Staubli VAL3: connectHostRos.pjx

--- connectHostRos.pjx ---
Parameters version=s7.9.1 stackSize=5000 millimeterUnit=true
Program file=decodeRecvData.pgx
Program file=encodeSendData.pgx
Program file=initTcpIpSocket.pgx
Program file=recvData.pgx
Program file=recvRosMsg.pgx
Program file=sendData.pgx
Program file=sendFbkMsg.pgx
Program file=start.pgx
Program file=stop.pgx
Data file=connectHostRos.dtx
Type name=FlagStatus path=Disk://RobotController_Libs/FlagStatus/FlagStatus.pjx
Type name=RobotStatus path=Disk://RobotController_Libs/RobotStatus/RobotStatus.pjx
Type name=CommParameter path=Disk://RobotController_Libs/CommParameter/CommParameter.pjx

--- connectHostRos.dtx ---
mdesc mNomSpeed
public sio soTcpIpFbk
public sio siTcpIpMotion
public num nRecvData[53]
public CommParameter cRosMotionParm
  [0]
    num port
    string target
    num clients
    num endOfString
    num timeOut
    num baudRate
    string parity
    num bits
    num stopBits
    string mode
    string flowControl
    bool nagle
public CommParameter cRosFbkParm
  [0]
    num port
    string target
    num clients
    num endOfString
    num timeOut
    num baudRate
    string parity
    num bits
    num stopBits
    string mode
    string flowControl
    bool nagle
public FlagStatus fRosStatus
  [0]
    num ForceFlag
    num RosFlag
    num RobotFlag
public num nSendData[52]

--- decodeRecvData.pgx ---
public program decodeRecvData(num& x_nRecvData[], RobotStatus& x_rRobotStatus, FlagStatus& x_fDataStatus, num& x_nRosFlagCmd)
  local num l_nNum
begin

  //This program is used for decoding the received data from host ROS contorlller.

  //suppose the received data containing 1 identifier, 24 joint status 27 cartesian status and 1 ROS flag
  //and ensure the received data intact
  if size(x_nRecvData)==53
    //assert the received ROS massages OK
    x_fDataStatus.RosFlag=1
    //decode the received data to the format of robot controller(Staubli SRS format)
    x_rRobotStatus.jointSpace.JointPos.j1=x_nRecvData[1]
    x_rRobotStatus.jointSpace.JointPos.j2=x_nRecvData[2]
    x_rRobotStatus.jointSpace.JointPos.j3=x_nRecvData[3]
    x_rRobotStatus.jointSpace.JointPos.j4=x_nRecvData[4]
    x_rRobotStatus.jointSpace.JointPos.j5=x_nRecvData[5]
    x_rRobotStatus.jointSpace.JointPos.j6=x_nRecvData[6]

    x_rRobotStatus.cartesianSpace.CartesianPos.trsf.x=x_nRecvData[25]
    x_rRobotStatus.cartesianSpace.CartesianPos.trsf.y=x_nRecvData[26]
    x_rRobotStatus.cartesianSpace.CartesianPos.trsf.z=x_nRecvData[27]
    x_rRobotStatus.cartesianSpace.CartesianPos.trsf.rx=x_nRecvData[28]
    x_rRobotStatus.cartesianSpace.CartesianPos.trsf.ry=x_nRecvData[29]
    x_rRobotStatus.cartesianSpace.CartesianPos.trsf.rz=x_nRecvData[30]

    for l_nNum=0 to 5
      x_rRobotStatus.jointSpace.JointVel[l_nNum]=x_nRecvData[l_nNum+7]
      x_rRobotStatus.jointSpace.JointAccel[l_nNum]=x_nRecvData[l_nNum+13]
      x_rRobotStatus.jointSpace.JointForce[l_nNum]=x_nRecvData[l_nNum+19]

      x_rRobotStatus.cartesianSpace.CartesianVel[l_nNum]=x_nRecvData[l_nNum+31]
      x_rRobotStatus.cartesianSpace.CartesianAccel[l_nNum]=x_nRecvData[l_nNum+37]
      x_rRobotStatus.cartesianSpace.CartesianForce[l_nNum]=x_nRecvData[l_nNum+43]
    endFor

    x_rRobotStatus.cartesianSpace.CarteResVel=x_nRecvData[49]
    x_rRobotStatus.cartesianSpace.CarteResAccel=x_nRecvData[50]
    x_rRobotStatus.cartesianSpace.CarteResForce=x_nRecvData[51]
    x_nRosFlagCmd=x_nRecvData[52]

  else
    x_fDataStatus.RosFlag=-1

  endIf

end

--- encodeSendData.pgx ---
public program encodeSendData(num& x_nSendData[], RobotStatus& x_rRobotStatus)
  local num l_nNum
begin

  //This program is used for encoding the data sent to the host ROS controller.

  //suppose the sent data containing 1 identifier，24 joint status and 27 cartesian status
  //and ensure the sent data intact
  x_nSendData[0]=0

  x_nSendData[1]=x_rRobotStatus.jointSpace.JointPos.j1
  x_nSendData[2]=x_rRobotStatus.jointSpace.JointPos.j2
  x_nSendData[3]=x_rRobotStatus.jointSpace.JointPos.j3
  x_nSendData[4]=x_rRobotStatus.jointSpace.JointPos.j4
  x_nSendData[5]=x_rRobotStatus.jointSpace.JointPos.j5
  x_nSendData[6]=x_rRobotStatus.jointSpace.JointPos.j6

  x_nSendData[25]=x_rRobotStatus.cartesianSpace.CartesianPos.trsf.x
  x_nSendData[26]=x_rRobotStatus.cartesianSpace.CartesianPos.trsf.y
  x_nSendData[27]=x_rRobotStatus.cartesianSpace.CartesianPos.trsf.z
  x_nSendData[28]=x_rRobotStatus.cartesianSpace.CartesianPos.trsf.rx
  x_nSendData[29]=x_rRobotStatus.cartesianSpace.CartesianPos.trsf.ry
  x_nSendData[30]=x_rRobotStatus.cartesianSpace.CartesianPos.trsf.rz

  for l_nNum=0 to 5
    x_nSendData[l_nNum+7]=x_rRobotStatus.jointSpace.JointVel[l_nNum]
    x_nSendData[l_nNum+13]=x_rRobotStatus.jointSpace.JointAccel[l_nNum]
    x_nSendData[l_nNum+19]=x_rRobotStatus.jointSpace.JointForce[l_nNum]

    x_nSendData[l_nNum+31]=x_rRobotStatus.cartesianSpace.CartesianVel[l_nNum]
    x_nSendData[l_nNum+37]=x_rRobotStatus.cartesianSpace.CartesianAccel[l_nNum]
    x_nSendData[l_nNum+43]=x_rRobotStatus.cartesianSpace.CartesianForce[l_nNum]
  endFor

  x_nSendData[49]=x_rRobotStatus.cartesianSpace.CarteResVel
  x_nSendData[50]=x_rRobotStatus.cartesianSpace.CarteResAccel
  x_nSendData[51]=x_rRobotStatus.cartesianSpace.CarteResForce

end

--- recvData.pgx ---
public program recvData(sio& x_sSioSocket, num& x_nRecvData[], RobotStatus& x_rRobotStatus, FlagStatus& x_fDataStatus, num& x_nRosFlagCmd)
  local num l_nRecvNum
begin

  //This program is used for receiving data from the host ROS controller.
  l_nRecvNum=sioGet(x_sSioSocket,x_nRecvData)
  if l_nRecvNum>0
    //call the decodeRecvData function to parse the received data
    call decodeRecvData(x_nRecvData,x_rRobotStatus,x_fDataStatus,x_nRosFlagCmd)
  endIf

end

--- recvRosMsg.pgx ---
public program recvRosMsg(RobotStatus& x_rRobotStatus, FlagStatus& x_fRosStatus, num x_nRosFlagCmd)
begin

  //This program is used for receiving motion planning command from the Host ROS controller and
  //ensuring the received ros massages correct.

  while true
    //Call the receive data function
    call recvData(siTcpIpMotion,nRecvData,x_rRobotStatus,x_fRosStatus,x_nRosFlagCmd)

    //Froce an end to the current task and enter the next sequence loop
    delay(0.0)

  endWhile

end

--- sendData.pgx ---
public program sendData(sio& x_sSioSocket, num& x_nSendData[], RobotStatus& x_rRobotStatus, FlagStatus& x_fDataStatus)
  local num l_nSendNum
begin

  //This program is used for sending the feedback data to the host ROS contorller.

  //call the encodeSendData function to encrypt the sent data
  call encodeSendData(x_nSendData,x_rRobotStatus)

  //send the encrypted data to the host ROS controller
  l_nSendNum=sioSet(x_sSioSocket,x_nSendData)
  if l_nSendNum==52
    x_fDataStatus.RosFlag=1
  else
    x_fDataStatus.RosFlag=-1
  endIf

end
